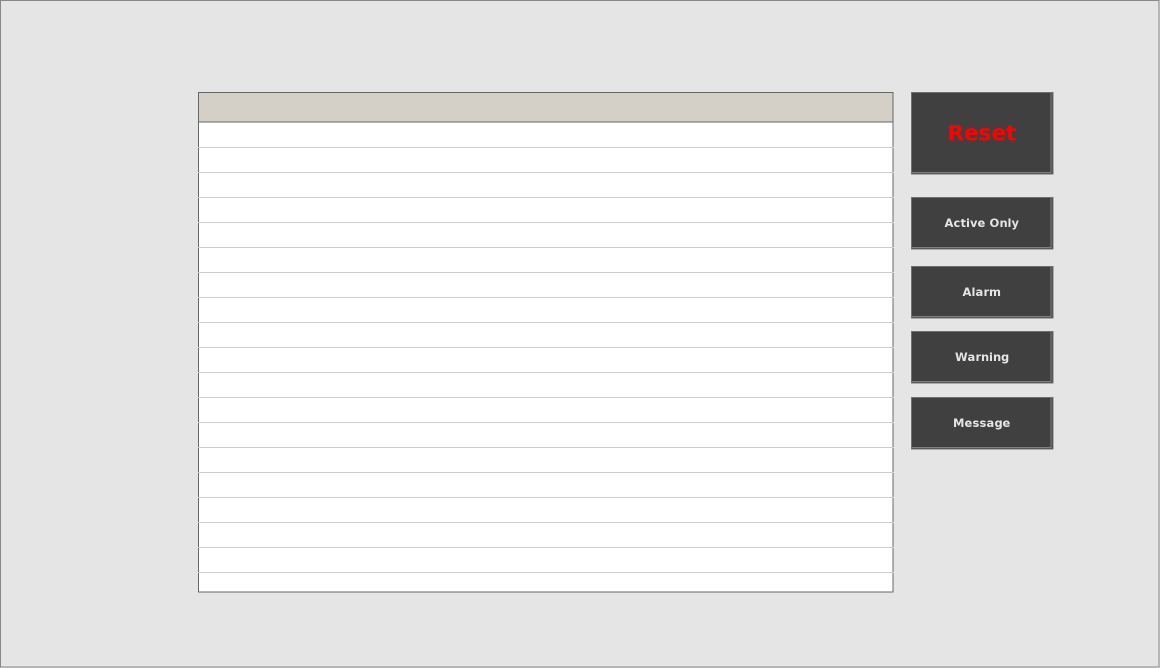
VISUALIZATION V_EventsHistoricalSimple  // 1160x668
    Table (198,92 695x500), data array: GVL_EHS.arrEventVisu
        p3854506369: GVL_EHS.arrEventVisu[INDEX].dwID
        p505689113: Date End
        p1218418051: GVL_EHS.arrEventVisu[INDEX].dtDateEnd
        p2237128397: Date Begin
        p3723444502: GVL_EHS.arrEventVisu[INDEX].dtDateBegin
        p511219082: Class
        p1892666644: GVL_EHS.arrEventVisu[INDEX].dwClass
        p1755163831: Message
        p338671338: GVL_EHS.arrEventVisu[INDEX].wsMessage
        p4092479075: Param
        p2170511999: GVL_EHS.arrEventVisu[INDEX].dwParam
        Columns.Column.[4].Template: GVL_EHS.arrEventVisu[INDEX].dwColor
        Columns.Column.[2].Template: GVL_EHS.arrEventVisu[INDEX].dwColor
        Columns.Column.[1].Template: GVL_EHS.arrEventVisu[INDEX].dwColor
        Columns.Column.[0].Template: GVL_EHS.arrEventVisu[INDEX].dwColor
        Columns.Column.[3].Template: GVL_EHS.arrEventVisu[INDEX].dwColor
        Columns.Column.[5].Template: GVL_EHS.arrEventVisu[INDEX].dwColor
    Button (911,197 142x52), "Active Only", colour toggle: P_EventsVisu.bFilterActiveOnly
        toggle P_EventsVisu.bFilterActiveOnly
    Button (911,92 142x82), "Reset"
    Button (911,266 142x52), "Alarm"
        tap GVL_HMI.bAlarm
    Button (911,331 142x52), "Warning"
        tap GVL_HMI.bWarning
    Button (911,397 142x52), "Message"
        tap GVL_HMI.bMessage
END_VISUALIZATION

(* stored: Version 1.1.0.1, ProductVersion 3.1.4024.3
   Visu V_EventsHistoricalSimple: Id {890e081a-3eb6-4af3-90c3-99fe0604e66c} *)
